FUNCTION_BLOCK FB_MotionDrive IMPLEMENTS I_MotionDrive
VAR
    {attribute 'hide'}
    iMoveRequest : I_MoveRequest;
    {attribute 'hide'}
    iEpicsMotionParamsStatus : I_EpicsMotionParamsStatus;
    {attribute 'hide'}
    iMotionAxis: I_MotionAxis;
    iMotionAxisDS402: I_MotionAxisDS402;
    {attribute 'hide'}
    iBrake 				: I_Brake;
    {attribute 'hide'}
    iMotionInterlocks	: I_MotionInterlocks;
    {attribute 'hide'}
    iMotionLogger 		: I_MotionLogger;
	iMotionDriveStateMachine : I_MotionDriveStateMachine;

    sName : STRING;

	bError: BOOL;
	nErrorId: UDINT;
	sErrorMessage: T_MAXSTRING;

	rtReset: R_TRIG;
	rtResetDone: R_TRIG;
	ftStop: F_TRIG;
END_VAR

// Restore axis parameters pass in a struct ref of parameters to restore
iMoveRequest.RestoreSettings(
	RestoreDone:=iMotionAxis.Status.bRestoreDone, 
	SavedPosition:=iMotionAxis.Status.fSavedPosition
);

// catch high priority message
// an extended error message from FB_MotionLogger will display cyclic errors and warning
IF iMotionAxis.Status.bError THEN
	bError := iMotionAxis.Status.bError;
	nErrorId := iMotionAxis.Status.nErrorID;
	sErrorMessage:= iMotionAxis.Status.sMessage;
ELSIF iMotionInterlocks.Error THEN
	bError := iMotionInterlocks.Error;
	nErrorId := iMotionInterlocks.ErrorID;
	sErrorMessage:= iMotionInterlocks.Message; 
// Warnings have lowest priority
ELSIF iMotionInterlocks.Warning THEN
	sErrorMessage:= iMotionInterlocks.Message; 
END_IF

iMoveRequest.MoveRequestError(
	Error := bError,
	ErrorId :=nErrorId,
	ErrorMessage:=sErrorMessage
);

// Forward Power block enable flags
iMotionAxis.Power(
	Enable:=iMotionInterlocks.PowerEnabled,
	Enable_Positive:=iMotionInterlocks.MoveForwardEnabled,
	Enable_Negative:=iMotionInterlocks.MoveBackwardEnabled,
    Override	:= 100.0,
    BufferMode	:= MC_Aborting
);

// Halt the Move
ftStop(CLK:=iMoveRequest.PauseMoveRequest(Busy:=iMotionAxis.Status.bBusy));
IF ftStop.Q THEN
	iMotionAxis.Halt(Deceleration:=iMoveRequest.Status.fDeceleration);
END_IF

// Reset
rtReset(CLK:=iMoveRequest.Status.bReset);
rtResetDone(CLK:=iMotionAxis.Status.bResetDone);
IF rtReset.Q THEN
   // Forward general reset event
   iMotionAxis.Reset();
 ELSIF rtResetDone.Q THEN
	// Reset EPICS ENbale, disbale drive power.
	iMoveRequest.ResetMoveEnable();
END_IF

iMotionInterlocks.AxisStatus(
      	HomeBusy:=iMotionAxis.Status.bHomeBusy,
      	PositiveDirection:=iMotionAxis.Status.bPositiveMotionIsEnabled,
       	NegativeDirection:=iMotionAxis.Status.bNegativeMotionIsEnabled 
);

//
iMoveRequest.MoveRequest(
	EnableDone:=iMotionAxis.AxisEnabled(),
	MoveOk:=iMotionInterlocks.MoveOk
);

// Forward drive commands to interlock blocks
iMotionInterlocks.DriveCommands(	
	Enable:= iMoveRequest.Status.bEnable,
	NewMoveReq:=iMoveRequest.Status.bNewMoveReq, 
	Reset:=iMotionAxis.Status.bResetDone
);


// Drive state machine
iMotionDriveStateMachine.StateMachine(	
		InterlockEvent:= iMotionInterlocks.InterlockEvent,
		Error	:=bError
);
						
// Forward axis state to brake FB
iBrake.AxisState := iMotionAxis.Status.eAxisState;

// Read Axis Parameter
iMotionAxis.ReadAxisParams(
	Enable:=TRUE, 
	RefreshDelay:=T#1S
);

// Save and Restore
iMotionAxis.SaveAxisParams(Enable:=TRUE);

// update EPICS status
iEpicsMotionParamsStatus.MotionParamsAndStatus( 
	PowerEnabled := iMotionInterlocks.PowerEnabled,
    PowerIsEnabled := iMotionAxis.Status.bPowerIsEnabled,
    Execute := iMoveRequest.Status.bExecute,
    LimHome := iMotionInterlocks.LimHome,
    MoveBackwardEnabled := iMotionInterlocks.MoveBackwardEnabled,
    MoveForwardEnabled := iMotionInterlocks.MoveForwardEnabled,
    MeasuredPositionDiff := iMotionAxis.Status.fMeasuredPositionDiff,
    MeasuredPosition := iMotionAxis.Status.fMeasuredPosition,
    MeasuredVelocity := iMotionAxis.Status.fMeasuredVelocity,
    PowerOverride := iMotionAxis.Status.fPowerOverride,
    Busy := iMotionAxis.Status.bBusy,
    HomeDone := iMotionAxis.Status.bHomeDone,
	MotionAxisId:=iMotionAxis.Status.nAxisId
);

METHOD PUBLIC CallAfterInit
VAR_INPUT
    iBrake : I_Brake;
    iMotionInterlocks : I_MotionInterlocks;
    iMotionLogger : I_MotionLogger;
    iMotionAxis: I_MotionAxis;
    iMoveRequest : I_MoveRequest;
    iEpicsMotionParamsStatus : I_EpicsMotionParamsStatus;
	iMotionDriveStateMachine : I_MotionDriveStateMachine;
END_VAR
THIS^.iMotionAxis := iMotionAxis;
THIS^.iMotionLogger:=iMotionLogger;
THIS^.iBrake:=iBrake;
THIS^.iMotionInterlocks:=iMotionInterlocks;
THIS^.iMoveRequest :=iMoveRequest;
THIS^.iEpicsMotionParamsStatus := iEpicsMotionParamsStatus;
THIS^.iMotionDriveStateMachine := iMotionDriveStateMachine;
END_METHOD

//FB_Init is always available implicitly and it is used primarily for initialization.
//The return value is not evaluated. For a specific influence, you can also declare the
//methods explicitly and provide additional code there with the standard initialization
//code. You can evaluate the return value.
METHOD FB_Init: BOOL
VAR_INPUT
    bInitRetains: BOOL; // TRUE: the retain variables are initialized (reset warm / reset cold)
    bInCopyCode: BOOL;  // TRUE: the instance will be copied to the copy code afterward (online change)
    iBrake : I_Brake;
    iMotionInterlocks : I_MotionInterlocks;
    iMotionLogger : I_MotionLogger;
    iMotionAxis: I_MotionAxis;
    iMoveRequest : I_MoveRequest;
    iEpicsMotionParamsStatus : I_EpicsMotionParamsStatus;
	iMotionDriveStateMachine : I_MotionDriveStateMachine;
END_VAR
THIS^.iMotionAxis := iMotionAxis;
THIS^.iMotionLogger:=iMotionLogger;
THIS^.iBrake:=iBrake;
THIS^.iMotionInterlocks:=iMotionInterlocks;
THIS^.iMoveRequest :=iMoveRequest;
THIS^.iEpicsMotionParamsStatus := iEpicsMotionParamsStatus;
THIS^.iMotionDriveStateMachine := iMotionDriveStateMachine;
END_METHOD

END_FUNCTION_BLOCK

(* stored: Version 1.1.0.1
   POU FB_MotionDrive: Id {60d91316-04e3-4af1-aaa1-6a890af932f7}, SpecialFunc None
   Method CallAfterInit: Id {f39ddf47-4815-43e7-8049-e534fb9f6092}
   Method FB_Init: Id {927f7c72-9006-42d1-8ac3-5d4ce66d6511} *)
